FUNCTION_BLOCK FB_Lesen EXTENDS FB_Basis
VAR_INPUT
	Reaktor			:I_Reaktor;
END_VAR

VAR_OUTPUT
END_VAR

VAR
END_VAR

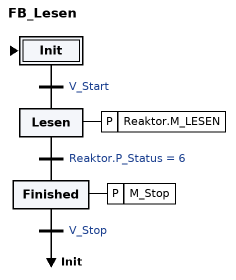
INITIAL_STEP Init:
END_STEP
TRANSITION FROM Init TO Lesen
    := V_Start;
END_TRANSITION
STEP Lesen:
    Reaktor.M_LESEN(P);
END_STEP
TRANSITION FROM Lesen TO Finished
    := Reaktor.P_Status = 6;
END_TRANSITION
STEP Finished:
    M_Stop(P);
END_STEP
TRANSITION FROM Finished TO Init
    := V_Stop;
END_TRANSITION

END_FUNCTION_BLOCK

(* stored: Version 1.1.0.1, ProductVersion 3.1.4024.12
   POU FB_Lesen: Id {a9f2d58b-2e85-46d4-bf1b-d8dc144c5b71}, SpecialFunc None *)
